FUNCTION_BLOCK Fraction EXTENDS SM_Fraction
VAR_INPUT
END_VAR
VAR_OUTPUT
END_VAR
VAR
    _testVar_Fraction : BOOL;
END_VAR

SUPER^();

END_FUNCTION_BLOCK

(* stored: Version 1.1.0.1, ProductVersion 3.1.4018.2
   POU Fraction: Id {7f7a3b46-710e-4911-8fea-f5c9d1ea3e27}, SpecialFunc None *)
